# EPICS StreamDevice protocol: streamDevice/keily.proto
# Keily's Sidekick EPICS protocol file
# Built by examining examples at: https://paulscherrerinstitute.github.io/StreamDevice/protocol.html#gen

Terminator = CR LF;

info {
	ExtraInput = Ignore;
	out "*IDN?";
	in "%39c";
}

debug {
   ExtraInput = Ignore;
   out "%s";
   in "%39c";
}

DisplayOnQ {
	out "DISPlay:ON?";
    in "%i";
}

DisplayText {
	out "DISPlay:TEXT %s";
}
